FUNCTION FC_Voltage0_10Raw_TO_Percentage : REAL
VAR_INPUT
	i : INT;
END_VAR
VAR
	f : REAL;
	nIntMax : INT := 32767;
	nIntMin : INT := 0;
END_VAR

FC_Voltage0_10Raw_TO_Percentage := 100*INT_TO_REAL(i-nIntMin)/(nIntMax-nIntMin);

END_FUNCTION

(* stored: Version 1.1.0.1, ProductVersion 3.1.4024.0
   POU FC_Voltage0_10Raw_TO_Percentage: Id {3c477724-9db8-4201-94ab-bbcc427d8baf}, SpecialFunc None *)
